SUBAPPLICATION SubscribeEventOpcUaPartial (* Publish event using OpcUa. The consumer is encapsulated *)
  (* Standard: 61499-2; Description: Copyright (c) 2019 fortiss GmbH This program and the accompanying materials are made SPDX-License-Identifier: EPL-2.0 *)
  (* Version 1.0, 2019-11-12, Jose Cabral, fortiss GmbH *)
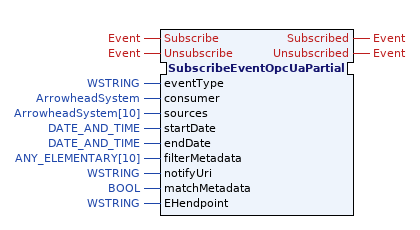
  EVENT_INPUT
    Subscribe;
    Unsubscribe;
  END_EVENT
  EVENT_OUTPUT
    Subscribed;
    Unsubscribed;
  END_EVENT
  VAR_INPUT
    eventType : WSTRING; (* Event type, similar to topics in MQTT *)
    consumer : ArrowheadSystem; (* The Subscriber ArrowheadSystem, that will consume the new events *)
    sources : ARRAY [0..9] OF ArrowheadSystem; (* List of ArrowheadSystem the Subscriber wants to receive events from *)
    startDate : DATE_AND_TIME; (* If set, the Subscriber wants to receive events with timestamps after this date-time *)
    endDate : DATE_AND_TIME; (* If set, the Subscriber wants to receive events with timestamps before this date-time *)
    filterMetadata : ARRAY [0..9] OF ANY_ELEMENTARY; (* Metadata about the events, which can be used for further filtering in format key=value *)
    notifyUri : WSTRING; (* The URL subpath where the Event Handler should sent the new events to *)
    matchMetadata : BOOL; (* Should the Event Handler filter events based on the metadata *)
    EHendpoint : WSTRING; (* Endpoint (IP:PORT/URI) of the Service Registry (not officially in the documentation, but it simplifies the FBs) *)
  END_VAR
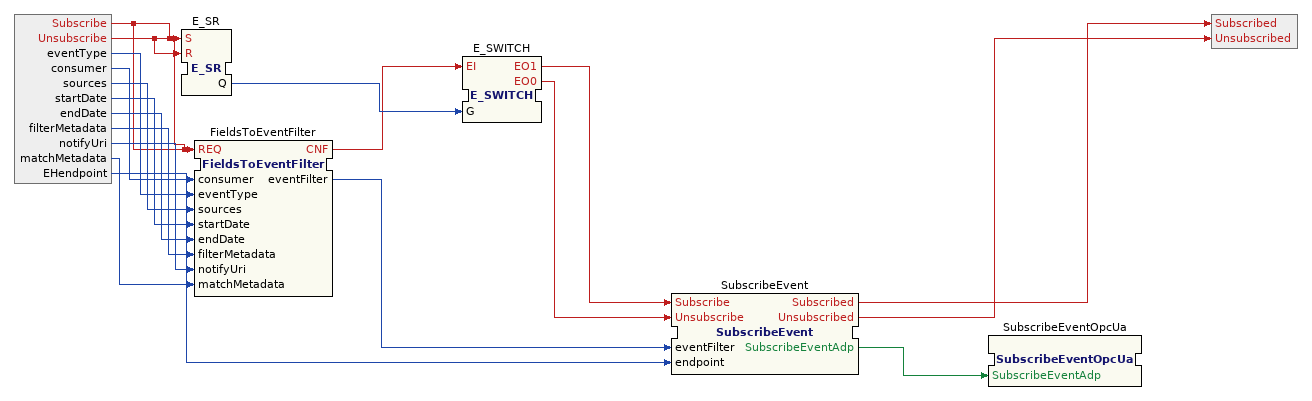
  FBS
    SubscribeEvent : SubscribeEvent;
    FieldsToEventFilter : FieldsToEventFilter;
    E_SWITCH : E_SWITCH;
    E_SR : E_SR;
    SubscribeEventOpcUa : SubscribeEventOpcUa;
  END_FBS
  EVENT_CONNECTIONS
    SubscribeEvent.Subscribed TO Subscribed;
    Subscribe TO FieldsToEventFilter.REQ;
    Unsubscribe TO FieldsToEventFilter.REQ;
    Subscribe TO E_SR.S;
    Unsubscribe TO E_SR.R;
    FieldsToEventFilter.CNF TO E_SWITCH.EI;
    E_SWITCH.EO1 TO SubscribeEvent.Subscribe;
    E_SWITCH.EO0 TO SubscribeEvent.Unsubscribe;
    SubscribeEvent.Unsubscribed TO Unsubscribed;
  END_CONNECTIONS
  DATA_CONNECTIONS
    FieldsToEventFilter.eventFilter TO SubscribeEvent.eventFilter;
    consumer TO FieldsToEventFilter.consumer;
    eventType TO FieldsToEventFilter.eventType;
    sources TO FieldsToEventFilter.sources;
    startDate TO FieldsToEventFilter.startDate;
    endDate TO FieldsToEventFilter.endDate;
    filterMetadata TO FieldsToEventFilter.filterMetadata;
    notifyUri TO FieldsToEventFilter.notifyUri;
    matchMetadata TO FieldsToEventFilter.matchMetadata;
    EHendpoint TO SubscribeEvent.endpoint;
    E_SR.Q TO E_SWITCH.G;
  END_CONNECTIONS
  ADAPTER_CONNECTIONS
    SubscribeEvent.SubscribeEventAdp TO SubscribeEventOpcUa.SubscribeEventAdp;
  END_CONNECTIONS
END_SUBAPPLICATION
